ABB RobotStudio station: Proyecto.rsstnx

Station Proyecto (saved by RobotStudio 23.2.10395.0)
Controller IRB140_6_81
  mechanical unit ROB_1: IRB140_6_81_C_03, 6 joints, base frame (0, 0, 0) mm
Layout (positions relative to the parent item):
  - IRB140_6_81_C_03 [mechanism, from %ABB.RobotStudio.Models.IRB140%\IRB140_6_81_C_G_03.rslib] at (0, 0, 0) mm; joint values [0, 0, 0, 0, 0.5236, 0] (rad or m)
Targets, tools, work objects and paths stored in the station, written as RAPID:
! task T_ROB1
MODULE Module1
  CONST robtarget Target_10:=[[466.539953566,-142.635568483,482.286643786],[0.280895683,0.141722572,0.948287929,-0.041980138],[-1,0,-1,0],[9E+09,9E+09,9E+09,9E+09,9E+09,9E+09]];
  CONST robtarget Target_20:=[[506.291651246,0,679.5],[0.5,0,0.866025404,0],[0,0,0,0],[9E+09,9E+09,9E+09,9E+09,9E+09,9E+09]];
  PROC Rutina1()
    MoveJ Target_10,v1000,z100,tool0\WObj:=wobj0;
  ENDPROC
  PROC main()
    WaitDO A1,1;
    Rutina1;
    WaitDO A2,1;
    RutinaHome;
    WaitDO A3,1;
    Rutina1;
    WaitDO B1,1;
    RutinaHome;
    WaitDO B2,1;
    Rutina1;
    WaitDO B3,1;
    RutinaHome;
    WaitDO P1,1;
    Rutina1;
    WaitDO P2,1;
    RutinaHome;
    WaitDO P3,1;
    Rutina1;
    WaitDO A1,1;
    Rutina1;
  ENDPROC
  PROC RutinaHome()
    MoveJ Target_20,v1000,z100,tool0\WObj:=wobj0;
  ENDPROC
ENDMODULE

